(* Logix 5000 project; controller FRIST_EXAMPLE Emulate 5570 rev 19.11; software revision 19.01 *)

TASK MainTask (continuous, watchdog 500 ms) : MainProgram

MODULES
   Local : Emulate 5570 (ICP 2, rev 19.11)
       : 1756-IB32 (ICP 3, rev 3.1, Input RPI 20 ms)   // DG-INPUT
       : vendor 1 type 7 code 8 (ICP 4, rev 3.1, Output RPI 20 ms)
       : 1756-IF6I (ICP 5, rev 1.1, Input RPI 100 ms)
       : 1756-OF8 (ICP 6, rev 1.1, Output RPI 12 ms)
END_MODULES

VAR_GLOBAL   (* controller tags *)
   DESLIGA : ALIAS FOR Local:3:I.Data.0;
   LIGA : ALIAS FOR Local:3:I.Data.1;
   MOTOR1 : ALIAS FOR Local:4:O.Data.0;
END_VAR

PROGRAM MainProgram   (* main routine MainRoutine *)

ROUTINE MainRoutine   (* ladder *)
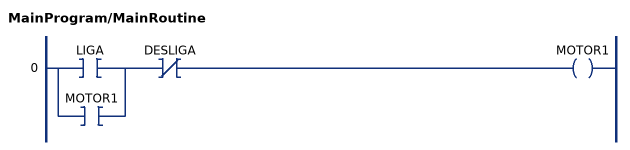
   0: [XIC(LIGA) ,XIC(MOTOR1) ]XIO(DESLIGA)OTE(MOTOR1);
END_ROUTINE
END_PROGRAM
